SUBAPPLICATION Licht (* Subapplication Type *)
  (* Standard: 61499-2 *)
  (* Version 1.0, 2023-01-29, Franz *)
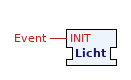
  EVENT_INPUT
    INIT; (* Service Initialization *)
  END_EVENT
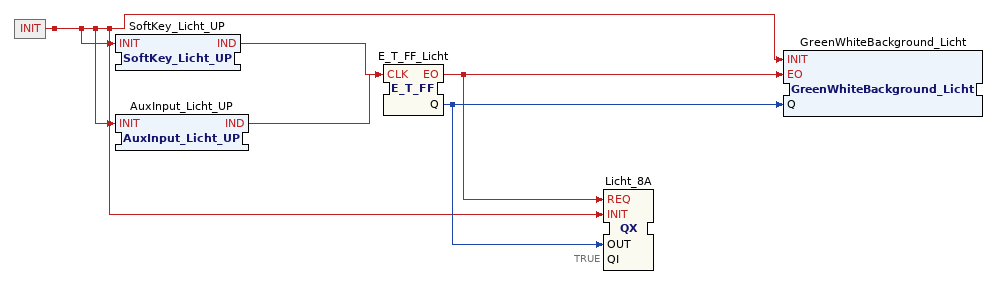
  FBS
    E_T_FF_Licht : E_T_FF;
    Licht_8A : QX(QI := TRUE);
  END_FBS
  SUBAPPS
    GreenWhiteBackground_Licht : GreenWhiteBackground_Licht;
    SoftKey_Licht_UP : SoftKey_Licht_UP;
    AuxInput_Licht_UP : AuxInput_Licht_UP;
  END_SUBAPPS
  EVENT_CONNECTIONS
    E_T_FF_Licht.EO TO Licht_8A.REQ;
    INIT TO GreenWhiteBackground_Licht.INIT;
    E_T_FF_Licht.EO TO GreenWhiteBackground_Licht.EO;
    INIT TO SoftKey_Licht_UP.INIT;
    SoftKey_Licht_UP.IND TO E_T_FF_Licht.CLK;
    INIT TO AuxInput_Licht_UP.INIT;
    AuxInput_Licht_UP.IND TO E_T_FF_Licht.CLK;
    INIT TO Licht_8A.INIT;
  END_CONNECTIONS
  DATA_CONNECTIONS
    E_T_FF_Licht.Q TO Licht_8A.OUT;
    E_T_FF_Licht.Q TO GreenWhiteBackground_Licht.Q;
  END_CONNECTIONS
END_SUBAPPLICATION
